TYPE "UDT_DI_Alarm_Conf"
VERSION : 0.2
// =============================================================================
// СТРУКТУРЫ ДЛЯ ДИСКРЕТНОГО АЛАРМА (FB_DI_Alarm)
// =============================================================================
   STRUCT
      En_Alarm { S7_SetPoint := 'True'} : Bool;   // 1 = Разрешение контроля аварии
      Invert { S7_SetPoint := 'True'} : Bool;   // 0 = NO (TRUE = Авария), 1 = NC (FALSE = Авария)
      Latch_Enable { S7_SetPoint := 'True'} : Bool;   // 1 = Фиксация аварии (требует сброса кнопкой Reset)
      Pad_Bit_3 { S7_SetPoint := 'True'} : Bool;   // Резерв
      Pad_Bit_4 { S7_SetPoint := 'True'} : Bool;   // Резерв
      Pad_Bit_5 { S7_SetPoint := 'True'} : Bool;   // Резерв
      Pad_Bit_6 { S7_SetPoint := 'True'} : Bool;   // Резерв
      Pad_Bit_7 { S7_SetPoint := 'True'} : Bool;   // Резерв
      Pad_Byte { S7_SetPoint := 'True'} : Byte;   // Выравнивание
      Delay { S7_SetPoint := 'True'} : Int := 1;   // Задержка срабатывания (в СЕКУНДАХ)
   END_STRUCT;

END_TYPE

